// TIA Portal V20 export
// export: Created 2026-07-12T13:33:04.9251016Z, ExportSetting WithDefaults, DisplayName Totally Integrated Automation Portal, DisplayVersion V20 Update 4, DisplayName TIA Portal Openness, DisplayVersion V20 Update 4, DisplayName TIA Portal Version Control Interface, DisplayVersion V20 Update 4, DisplayName STEP 7 Professional, DisplayVersion V20 Update 4, DisplayName STEP 7 Safety, DisplayVersion V20 Update 2, DisplayName WinCC Basic/Comfort/Advanced, DisplayVersion V20 Update 4, DisplayName WinCC Unified, DisplayVersion V20 Update 4
DATA_BLOCK "DB_Mesurements"   // DB13
{ S7_Optimized_Access := 'FALSE' }
VERSION : 0.1
// stored: AutoNumber true, IsOnlyStoredInLoadMemory false, IsWriteProtectedInAS false
   VAR RETAIN
      i_ThicknessRaw : Int;   // Encoder
      r_ThicknessScaled : Real;   // Encoder
      ProxyCount : DInt;   // Proximity
   END_VAR
BEGIN
END_DATA_BLOCK
